FUNCTION_BLOCK "fbArchiveParRectifier"
{ S7_Optimized_Access := 'TRUE' }
VERSION : 0.8
   VAR
      parRectifier : Array[1..1] of "tParameterRectifier";
   END_VAR

   VAR_TEMP
      tempInt : Int;
   END_VAR


BEGIN
END_FUNCTION_BLOCK

